% RSLogix 500 project CCHDUMP_backup_no_tags_eulises_feb_28_2020.RSS, saved by version 11.00.00.00 %
PROJECT "CCHDUMP"    % processor: MicroLogix 1200 %

PROGRAM FILES
  LAD 2   62 rungs

DATA FILES
  O0 OUTPUT  4 elements
  I1 INPUT  4 elements
  S2 STATUS  66 elements
  B3 BINARY  3 elements
  T4 TIMER  19 elements
  C5 COUNTER  1 elements
  R6 CONTROL  1 elements
  N7 INTEGER  1 elements
  F8 FLOAT  1 elements

LADDER 2
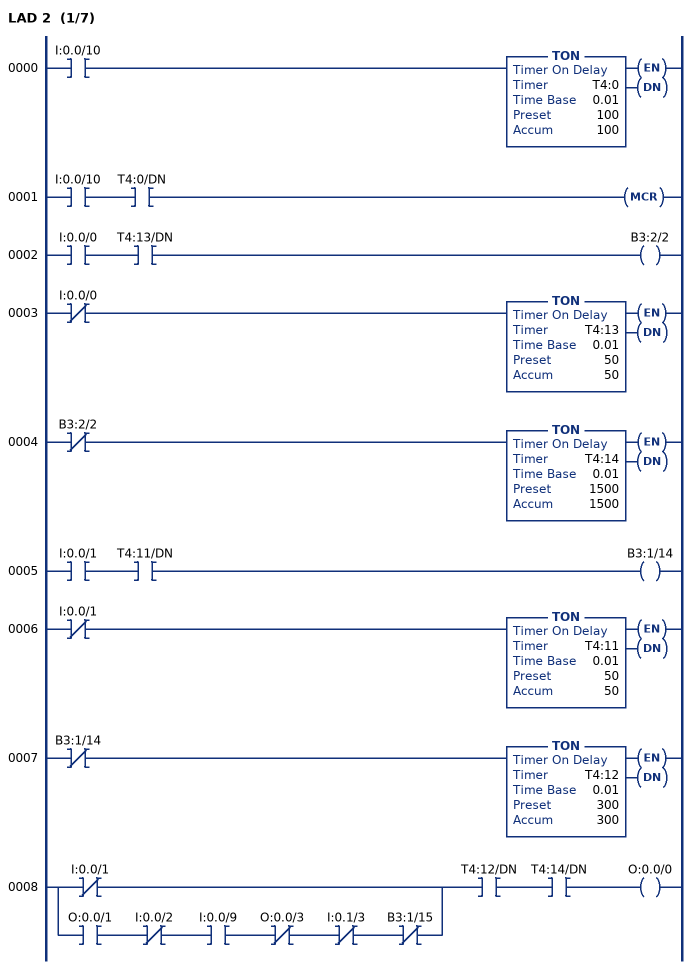
% Rung: 0 %
SOR XIC I:0.0/10 TON T4:0 0.01 100 100 EOR
% Rung: 1 %
SOR XIC I:0.0/10 XIC T4:0/DN MCR EOR
% Rung: 2 %
SOR XIC I:0.0/0 XIC T4:13/DN OTE B3:2/2 EOR
% Rung: 3 %
SOR XIO I:0.0/0 TON T4:13 0.01 50 50 EOR
% Rung: 4 %
SOR XIO B3:2/2 TON T4:14 0.01 1500 1500 EOR
% Rung: 5 %
SOR XIC I:0.0/1 XIC T4:11/DN OTE B3:1/14 EOR
% Rung: 6 %
SOR XIO I:0.0/1 TON T4:11 0.01 50 50 EOR
% Rung: 7 %
SOR XIO B3:1/14 TON T4:12 0.01 300 300 EOR
% Rung: 8 %
SOR BST XIO I:0.0/1 NXB XIC O:0.0/1 XIO I:0.0/2 XIC I:0.0/9 XIO O:0.0/3 XIO I:0.1/3 XIO B3:1/15 BND XIC T4:12/DN XIC T4:14/DN OTE O:0.0/0 EOR

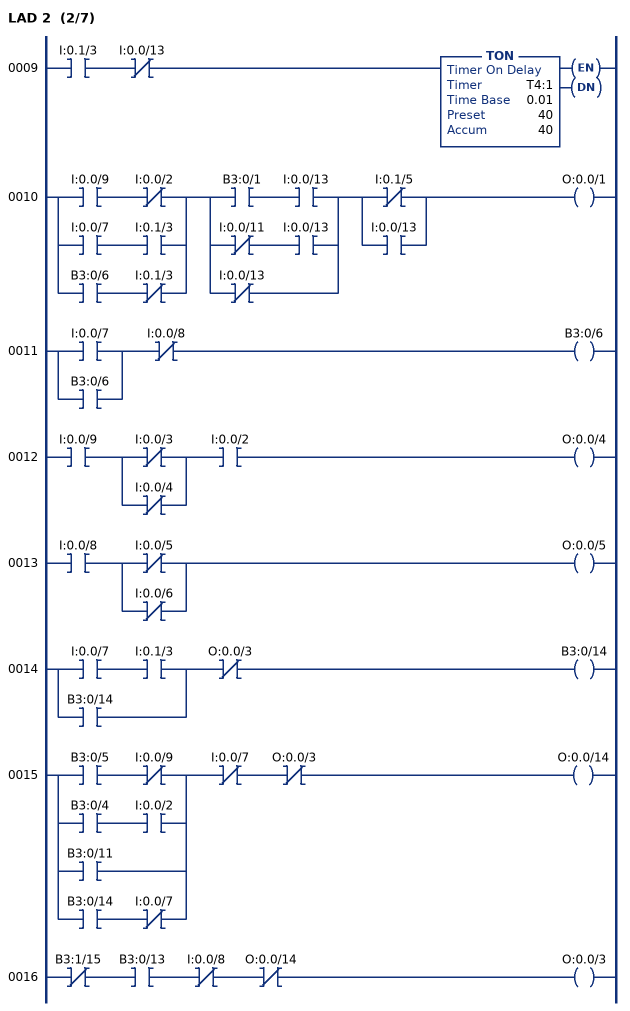
% Rung: 9 %
SOR XIC I:0.1/3 XIO I:0.0/13 TON T4:1 0.01 40 40 EOR
% Rung: 10 %
SOR BST XIC I:0.0/9 XIO I:0.0/2 NXB XIC I:0.0/7 XIC I:0.1/3 NXB XIC B3:0/6 XIO I:0.1/3 BND BST XIC B3:0/1 XIC I:0.0/13 NXB XIO I:0.0/11 XIC I:0.0/13 NXB XIO I:0.0/13 BND BST XIO I:0.1/5 NXB XIC I:0.0/13 BND OTE O:0.0/1 EOR
% Rung: 11 %
SOR BST XIC I:0.0/7 NXB XIC B3:0/6 BND XIO I:0.0/8 OTE B3:0/6 EOR
% Rung: 12 %
SOR XIC I:0.0/9 BST XIO I:0.0/3 NXB XIO I:0.0/4 BND XIC I:0.0/2 OTE O:0.0/4 EOR
% Rung: 13 %
SOR XIC I:0.0/8 BST XIO I:0.0/5 NXB XIO I:0.0/6 BND OTE O:0.0/5 EOR
% Rung: 14 %
SOR BST XIC I:0.0/7 XIC I:0.1/3 NXB XIC B3:0/14 BND XIO O:0.0/3 OTE B3:0/14 EOR
% Rung: 15 %
SOR BST XIC B3:0/5 XIO I:0.0/9 NXB XIC B3:0/4 XIC I:0.0/2 NXB XIC B3:0/11 NXB XIC B3:0/14 XIO I:0.0/7 BND XIO I:0.0/7 XIO O:0.0/3 OTE O:0.0/14 EOR
% Rung: 16 %
SOR XIO B3:1/15 XIC B3:0/13 XIO I:0.0/8 XIO O:0.0/14 OTE O:0.0/3 EOR

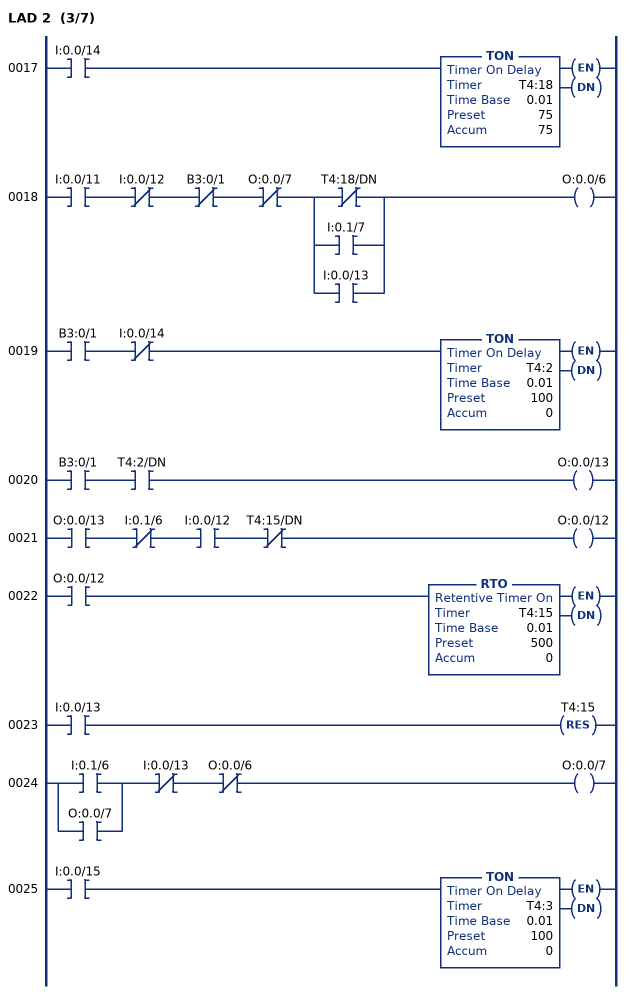
% Rung: 17 %
SOR XIC I:0.0/14 TON T4:18 0.01 75 75 EOR
% Rung: 18 %
SOR XIC I:0.0/11 XIO I:0.0/12 XIO B3:0/1 XIO O:0.0/7 BST XIO T4:18/DN NXB XIC I:0.1/7 NXB XIC I:0.0/13 BND OTE O:0.0/6 EOR
% Rung: 19 %
SOR XIC B3:0/1 XIO I:0.0/14 TON T4:2 0.01 100 0 EOR
% Rung: 20 %
SOR XIC B3:0/1 XIC T4:2/DN OTE O:0.0/13 EOR
% Rung: 21 %
SOR XIC O:0.0/13 XIO I:0.1/6 XIC I:0.0/12 XIO T4:15/DN OTE O:0.0/12 EOR
% Rung: 22 %
SOR XIC O:0.0/12 RTO T4:15 0.01 500 0 EOR
% Rung: 23 %
SOR XIC I:0.0/13 RES T4:15 EOR
% Rung: 24 %
SOR BST XIC I:0.1/6 NXB XIC O:0.0/7 BND XIO I:0.0/13 XIO O:0.0/6 OTE O:0.0/7 EOR
% Rung: 25 %
SOR XIC I:0.0/15 TON T4:3 0.01 100 0 EOR

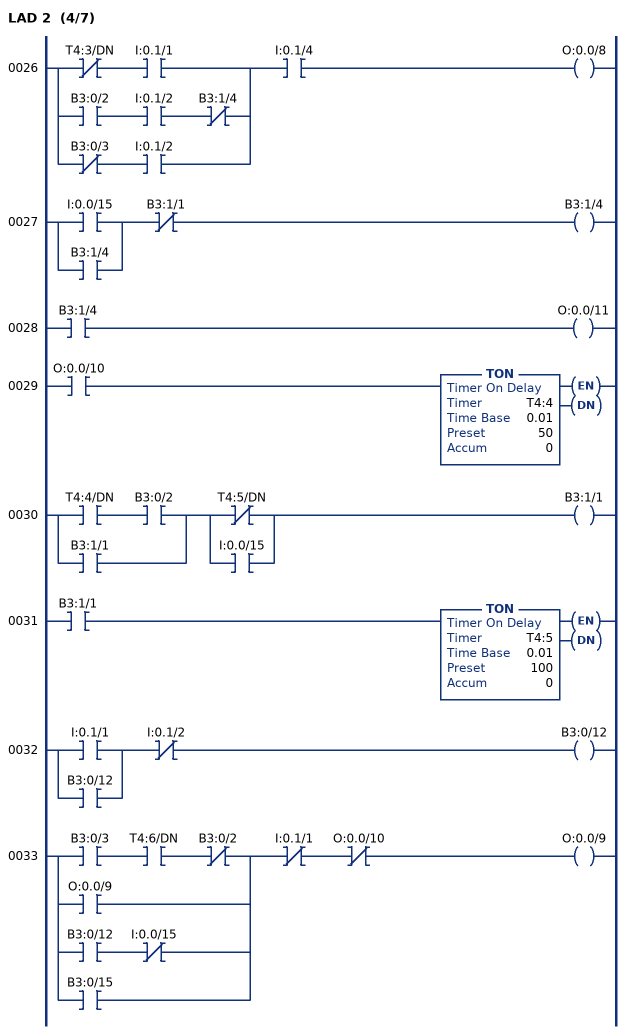
% Rung: 26 %
SOR BST XIO T4:3/DN XIC I:0.1/1 NXB XIC B3:0/2 XIC I:0.1/2 XIO B3:1/4 NXB XIO B3:0/3 XIC I:0.1/2 BND XIC I:0.1/4 OTE O:0.0/8 EOR
% Rung: 27 %
SOR BST XIC I:0.0/15 NXB XIC B3:1/4 BND XIO B3:1/1 OTE B3:1/4 EOR
% Rung: 28 %
SOR XIC B3:1/4 OTE O:0.0/11 EOR
% Rung: 29 %
SOR XIC O:0.0/10 TON T4:4 0.01 50 0 EOR
% Rung: 30 %
SOR BST XIC T4:4/DN XIC B3:0/2 NXB XIC B3:1/1 BND BST XIO T4:5/DN NXB XIC I:0.0/15 BND OTE B3:1/1 EOR
% Rung: 31 %
SOR XIC B3:1/1 TON T4:5 0.01 100 0 EOR
% Rung: 32 %
SOR BST XIC I:0.1/1 NXB XIC B3:0/12 BND XIO I:0.1/2 OTE B3:0/12 EOR
% Rung: 33 %
SOR BST XIC B3:0/3 XIC T4:6/DN XIO B3:0/2 NXB XIC O:0.0/9 NXB XIC B3:0/12 XIO I:0.0/15 NXB XIC B3:0/15 BND XIO I:0.1/1 XIO O:0.0/10 OTE O:0.0/9 EOR

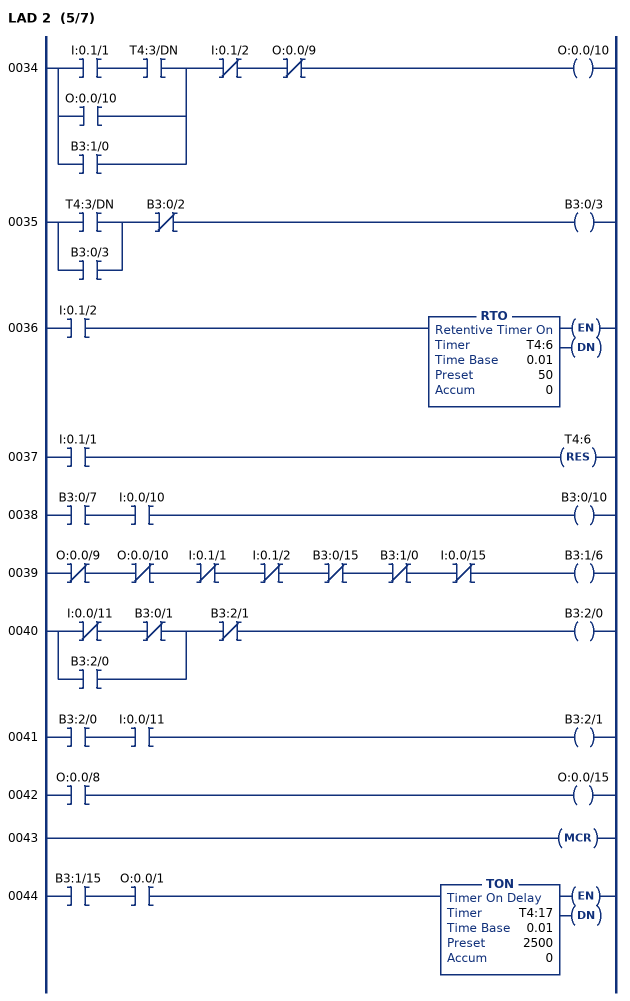
% Rung: 34 %
SOR BST XIC I:0.1/1 XIC T4:3/DN NXB XIC O:0.0/10 NXB XIC B3:1/0 BND XIO I:0.1/2 XIO O:0.0/9 OTE O:0.0/10 EOR
% Rung: 35 %
SOR BST XIC T4:3/DN NXB XIC B3:0/3 BND XIO B3:0/2 OTE B3:0/3 EOR
% Rung: 36 %
SOR XIC I:0.1/2 RTO T4:6 0.01 50 0 EOR
% Rung: 37 %
SOR XIC I:0.1/1 RES T4:6 EOR
% Rung: 38 %
SOR XIC B3:0/7 XIC I:0.0/10 OTE B3:0/10 EOR
% Rung: 39 %
SOR XIO O:0.0/9 XIO O:0.0/10 XIO I:0.1/1 XIO I:0.1/2 XIO B3:0/15 XIO B3:1/0 XIO I:0.0/15 OTE B3:1/6 EOR
% Rung: 40 %
SOR BST XIO I:0.0/11 XIO B3:0/1 NXB XIC B3:2/0 BND XIO B3:2/1 OTE B3:2/0 EOR
% Rung: 41 %
SOR XIC B3:2/0 XIC I:0.0/11 OTE B3:2/1 EOR
% Rung: 42 %
SOR XIC O:0.0/8 OTE O:0.0/15 EOR
% Rung: 43 %
SOR MCR EOR
% Rung: 44 %
SOR XIC B3:1/15 XIC O:0.0/1 TON T4:17 0.01 2500 0 EOR

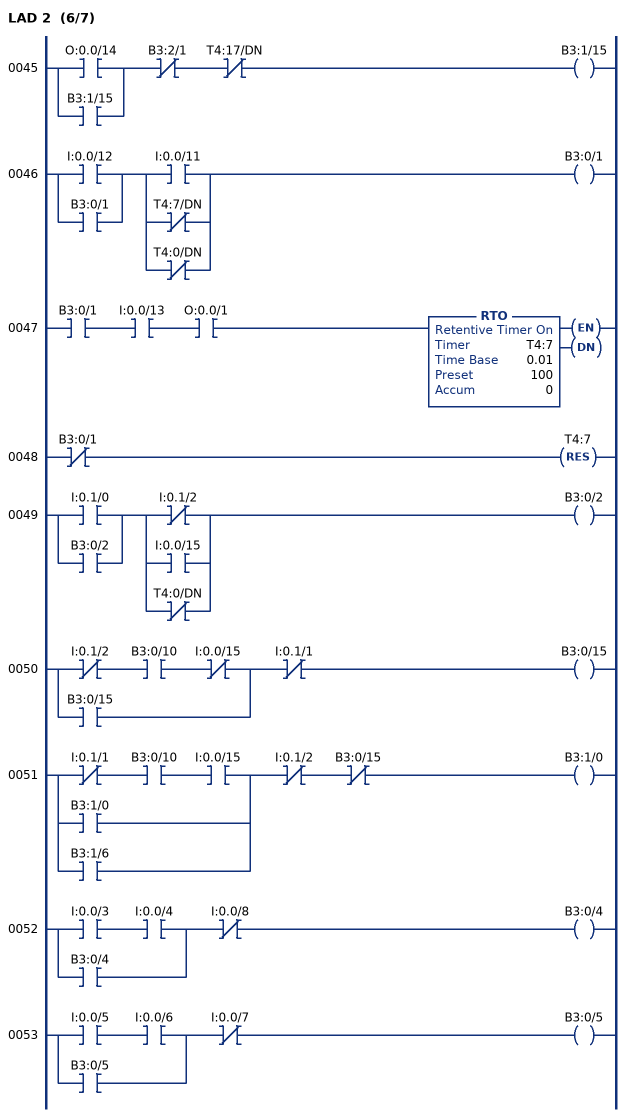
% Rung: 45 %
SOR BST XIC O:0.0/14 NXB XIC B3:1/15 BND XIO B3:2/1 XIO T4:17/DN OTE B3:1/15 EOR
% Rung: 46 %
SOR BST XIC I:0.0/12 NXB XIC B3:0/1 BND BST XIC I:0.0/11 NXB XIO T4:7/DN NXB XIO T4:0/DN BND OTE B3:0/1 EOR
% Rung: 47 %
SOR XIC B3:0/1 XIC I:0.0/13 XIC O:0.0/1 RTO T4:7 0.01 100 0 EOR
% Rung: 48 %
SOR XIO B3:0/1 RES T4:7 EOR
% Rung: 49 %
SOR BST XIC I:0.1/0 NXB XIC B3:0/2 BND BST XIO I:0.1/2 NXB XIC I:0.0/15 NXB XIO T4:0/DN BND OTE B3:0/2 EOR
% Rung: 50 %
SOR BST XIO I:0.1/2 XIC B3:0/10 XIO I:0.0/15 NXB XIC B3:0/15 BND XIO I:0.1/1 OTE B3:0/15 EOR
% Rung: 51 %
SOR BST XIO I:0.1/1 XIC B3:0/10 XIC I:0.0/15 NXB XIC B3:1/0 NXB XIC B3:1/6 BND XIO I:0.1/2 XIO B3:0/15 OTE B3:1/0 EOR
% Rung: 52 %
SOR BST XIC I:0.0/3 XIC I:0.0/4 NXB XIC B3:0/4 BND XIO I:0.0/8 OTE B3:0/4 EOR
% Rung: 53 %
SOR BST XIC I:0.0/5 XIC I:0.0/6 NXB XIC B3:0/5 BND XIO I:0.0/7 OTE B3:0/5 EOR

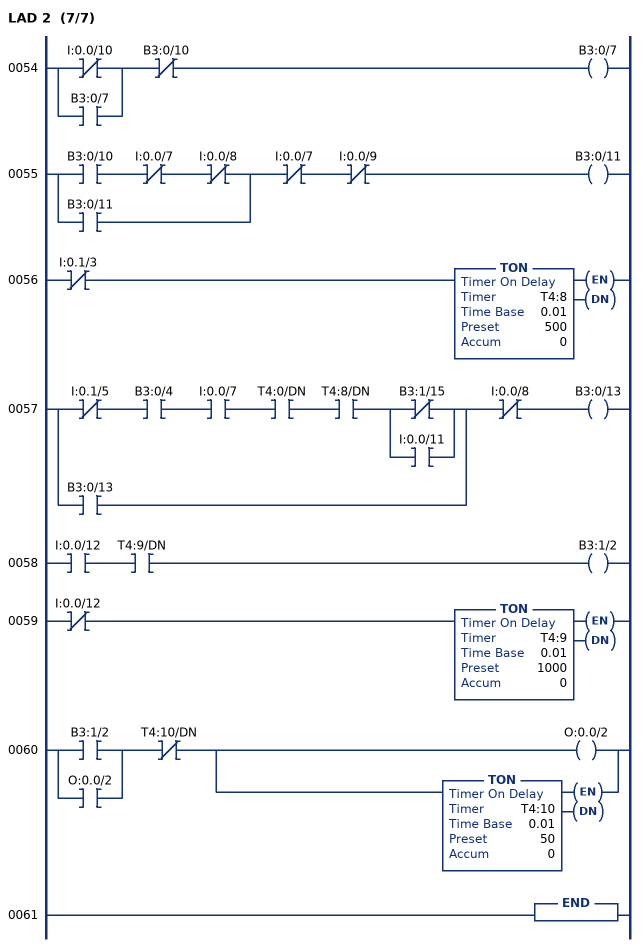
% Rung: 54 %
SOR BST XIO I:0.0/10 NXB XIC B3:0/7 BND XIO B3:0/10 OTE B3:0/7 EOR
% Rung: 55 %
SOR BST XIC B3:0/10 XIO I:0.0/7 XIO I:0.0/8 NXB XIC B3:0/11 BND XIO I:0.0/7 XIO I:0.0/9 OTE B3:0/11 EOR
% Rung: 56 %
SOR XIO I:0.1/3 TON T4:8 0.01 500 0 EOR
% Rung: 57 %
SOR BST XIO I:0.1/5 XIC B3:0/4 XIC I:0.0/7 XIC T4:0/DN XIC T4:8/DN BST XIO B3:1/15 NXB XIC I:0.0/11 BND NXB XIC B3:0/13 BND XIO I:0.0/8 OTE B3:0/13 EOR
% Rung: 58 %
SOR XIC I:0.0/12 XIC T4:9/DN OTE B3:1/2 EOR
% Rung: 59 %
SOR XIO I:0.0/12 TON T4:9 0.01 1000 0 EOR
% Rung: 60 %
SOR BST XIC B3:1/2 NXB XIC O:0.0/2 BND XIO T4:10/DN BST OTE O:0.0/2 NXB TON T4:10 0.01 50 0 BND EOR
% Rung: 61 %
SOR END EOR

DATA TABLE (non-zero values as saved)
DATA B3
% B3:0 % 0X1026 0X8010 0X0000
DATA T4
% .PRE .ACC %
% T4:0 % 100 100
% T4:1 % 40 40
% T4:2 % 100 0
% T4:3 % 100 0
% T4:4 % 50 0
% T4:5 % 100 0
% T4:6 % 50 0
% T4:7 % 100 0
% T4:8 % 500 0
% T4:9 % 1000 0
% T4:10 % 50 0
% T4:11 % 50 50
% T4:12 % 300 300
% T4:13 % 50 50
% T4:14 % 1500 1500
% T4:15 % 500 0
% T4:16 % 100 0
% T4:17 % 2500 0
% T4:18 % 75 75
